Yaskawa INFORM job: X2_55A(90,180).JBI

/JOB
//NAME X2_55A(90,180)
//POS
///NPOS 356,356,356,16,0,0
///TOOL 0
///POSTYPE PULSE
///PULSE
C00000=3109,-122452,-100913,-73,83322,449
C00001=-57547,-44507,-45529,-37768,86502,54365
C00002=-65928,-27646,-34572,-36764,84429,51561
C00003=-68932,-27355,-32037,-36417,82009,51120
C00004=-70133,-27145,-30956,-36281,81048,50940
C00005=-71251,-29014,-32241,-36126,80438,50675
C00006=-70937,-28647,-32231,-36159,80720,50713
C00007=-70939,-28348,-30359,-36244,79905,50983
C00008=-70850,-28266,-30689,-36235,80141,50942
C00009=-71777,-26040,-29151,-36077,79912,50630
C00010=-70850,-28266,-30689,-36235,80141,50942
C00011=-69640,-28520,-31799,-36368,81104,51127
C00012=-66609,-28920,-34410,-36705,83528,51580
C00013=-67283,-40522,-42778,-21836,57084,56863
C00014=-69666,-37175,-37764,-20920,55189,56238
C00015=-70593,-35779,-35703,-20558,54438,55990
C00016=-70595,-35399,-33785,-20806,53513,56182
C00017=-71439,-34878,-33636,-20299,53466,55818
C00018=-72039,-34449,-33357,-19958,53365,55574
C00019=-70600,-35459,-34012,-20775,53614,56158
C00020=-69673,-36879,-36092,-21134,54366,56408
C00021=-67291,-40287,-41153,-22043,56263,57036
C00022=-54757,-64654,-56678,-26574,55995,60610
C00023=-66125,-22240,-12046,-37767,75415,54591
C00024=-69120,-21153,-8852,-37720,72980,54160
C00025=-70318,-20628,-7503,-37704,72009,53986
C00026=-71434,-22405,-8777,-37615,71420,53709
C00027=-71106,-21887,-8483,-37633,71631,53777
C00028=-71108,-21030,-6132,-37829,70825,54070
C00029=-70936,-21522,-6647,-37833,70951,54100
C00030=-71862,-19395,-5114,-37710,70668,53794
C00031=-70936,-21522,-6647,-37833,70951,54100
C00032=-66696,-23294,-11311,-37869,74371,54717
C00033=-67477,-36863,-27706,-23811,50186,58383
C00034=-69851,-33011,-22248,-22972,48242,57743
C00035=-70774,-31410,-19999,-22642,47467,57490
C00036=-70776,-30665,-17785,-22990,46560,57721
C00037=-70660,-30833,-18099,-23019,46692,57745
C00038=-72095,-29866,-17454,-22146,46391,57112
C00039=-70660,-30833,-18099,-23019,46692,57745
C00040=-67358,-36360,-25881,-24167,49428,58637
C00041=-57529,-55156,-37288,-27679,48780,61381
C00042=-66162,-22086,-11962,-37760,75421,54573
C00043=-69154,-20998,-8767,-37712,72987,54143
C00044=-70350,-20473,-7417,-37696,72017,53969
C00045=-71465,-22250,-8693,-37606,71429,53692
C00046=-74636,-20949,-11222,-31484,73172,51606
C00047=-71188,-20903,-6014,-37823,70785,54049
C00048=-71042,-21313,-6495,-37820,70916,54065
C00049=-71965,-19182,-4958,-37697,70633,53761
C00050=-71042,-21313,-6495,-37820,70916,54065
C00051=-66808,-23094,-11168,-37857,74333,54682
C00052=-67549,-36655,-27551,-23768,50176,58352
C00053=-69918,-32800,-22087,-22931,48232,57713
C00054=-70839,-31198,-19836,-22602,47457,57461
C00055=-70841,-30454,-17622,-22950,46550,57692
C00056=-70807,-30574,-17946,-22919,46687,57673
C00057=-72239,-29602,-17296,-22048,46388,57041
C00058=-70807,-30574,-17946,-22919,46687,57673
C00059=-67516,-36108,-25740,-24067,49421,58563
C00060=-58006,-54475,-36914,-27392,48730,61159
C00061=-66150,-22232,-11999,-37769,75384,54591
C00062=-69146,-21141,-8802,-37722,72949,54160
C00063=-70343,-20614,-7451,-37706,71978,53986
C00064=-71460,-22391,-8725,-37617,71389,53709
C00065=-76354,-9489,-5358,-27324,81880,47708
C00066=-80283,-13253,-8650,-21924,78677,47540
C00067=-72863,-23243,-10183,-35045,70283,54216
C00068=-72091,-18996,-4868,-37675,70611,53714
C00069=-71171,-21130,-6410,-37799,70893,54017
C00070=-66943,-22922,-11092,-37839,74307,54632
C00071=-67592,-36530,-27454,-23743,50168,58333
C00072=-69958,-32673,-21987,-22907,48224,57696
C00073=-70878,-31070,-19735,-22578,47450,57444
C00074=-70881,-30326,-17520,-22926,46541,57675
C00075=-70888,-30451,-17880,-22864,46685,57634
C00076=-72318,-29476,-17227,-21993,46388,57002
C00077=-70888,-30451,-17880,-22864,46685,57634
C00078=-67602,-35989,-25679,-24012,49417,58523
C00079=-55368,-59030,-40465,-28749,49477,62233
C00080=-66281,-21711,-11569,-37757,75329,54554
C00081=-69266,-20611,-8362,-37710,72898,54126
C00082=-75255,-19909,-10818,-29439,72911,51436
C00083=-75255,-19389,-9203,-29543,72275,51605
C00084=-75255,-19909,-10818,-29439,72911,51436
C00085=-76150,-21069,-11659,-29326,72528,51179
C00086=-75255,-19909,-10818,-29439,72911,51436
C00087=-75952,-17840,-9303,-29323,72782,51192
C00088=-76627,-15764,-7759,-29212,72649,50956
C00089=-75952,-17840,-9303,-29323,72782,51192
C00090=-67008,-22654,-10922,-37828,74305,54605
C00091=-67726,-36243,-27274,-23659,50164,58271
C00092=-70084,-32383,-21799,-22824,48221,57636
C00093=-71001,-30778,-19544,-22496,47446,57385
C00094=-71004,-30035,-17329,-22843,46537,57615
C00095=-71019,-30169,-17685,-22780,46672,57573
C00096=-72445,-29190,-17028,-21910,46377,56942
C00097=-71019,-30169,-17685,-22780,46672,57573
C00098=-67743,-35714,-25496,-23926,49403,58459
C00099=-55737,-58548,-40210,-28536,49431,62065
C00100=-62068,-51424,-36574,-22006,75894,31841
C00101=-60714,-28502,-21418,-45365,79926,-4626
C00102=-66771,-18477,-14837,-68384,79212,-42474
C00103=-69189,-16510,-10390,-68595,76911,-42051
C00104=-70947,-14387,-8158,-68595,75621,-42165
C00105=-70947,-13867,-6433,-68771,75311,-41816
C00106=-70947,-14164,-7409,-68671,75485,-42013
C00107=-71934,-13328,-6772,-68630,74836,-42164
C00108=-70947,-14164,-7409,-68671,75485,-42013
C00109=-66757,-18118,-13479,-68487,78967,-42191
C00110=-63228,-11986,-9955,-68477,81724,-42141
C00111=-63445,-12696,-10506,-68473,81568,-42159
C00112=-66764,-18741,-15037,-68386,79212,-42468
C00113=-69186,-16774,-10592,-68597,76909,-42046
C00114=-70875,-13966,-7307,-68664,75547,-42021
C00115=-70875,-13696,-6414,-68755,75387,-41841
C00116=-70875,-13966,-7307,-68664,75547,-42021
C00117=-71778,-13120,-6662,-68624,74954,-42161
C00118=-70875,-13966,-7307,-68664,75547,-42021
C00119=-66661,-18411,-13691,-68493,79023,-42169
C00120=-63445,-12696,-10506,-68473,81568,-42159
C00121=-63865,-13952,-11469,-68464,81265,-42192
C00122=-66537,-18783,-15074,-68396,79365,-42438
C00123=-68961,-16831,-10641,-68604,77060,-42016
C00124=-70699,-13899,-7235,-68671,75661,-41992
C00125=-70699,-13580,-6183,-68778,75474,-41781
C00126=-70699,-13899,-7235,-68671,75661,-41992
C00127=-71619,-12932,-6499,-68632,75061,-42136
C00128=-70699,-13899,-7235,-68671,75661,-41992
C00129=-66539,-18412,-13687,-68498,79104,-42151
C00130=-63865,-13952,-11469,-68464,81265,-42192
C00131=-63260,-13360,-10989,-68484,81675,-42115
C00132=-66441,-19168,-15326,-68406,79413,-42406
C00133=-68872,-17218,-10898,-68615,77104,-41986
C00134=-70768,-14438,-7612,-68680,75597,-41981
C00135=-70768,-14095,-6488,-68794,75397,-41755
C00136=-70768,-14438,-7612,-68680,75597,-41981
C00137=-71628,-14065,-7329,-68648,75028,-42105
C00138=-70768,-14438,-7612,-68680,75597,-41981
C00139=-66448,-18790,-13996,-68502,79163,-42137
C00140=-63260,-13360,-10989,-68484,81675,-42115
C00141=-61191,-13759,-10892,-73705,82833,-41510
C00142=-64290,-19711,-15321,-73681,80576,-41688
C00143=-66947,-17907,-11278,-73881,78250,-41270
C00144=-68815,-15776,-8601,-73968,76784,-41217
C00145=-68815,-15434,-7486,-74073,76629,-40986
C00146=-68815,-15776,-8601,-73968,76784,-41217
C00147=-69853,-15286,-8234,-73951,76069,-41336
C00148=-68815,-15776,-8601,-73968,76784,-41217
C00149=-64280,-19397,-14090,-73763,80400,-41421
C00150=-61191,-13759,-10892,-73705,82833,-41510
C00151=-66549,4585,8841,-68757,84788,-39990
C00152=-68719,6226,13286,-68971,82600,-39461
C00153=-70299,8854,16372,-69091,81328,-39429
C00154=-70565,4457,12550,-69090,81182,-39506
C00155=-70671,1948,10411,-69092,81122,-39532
C00156=-70937,-1261,7725,-69102,80944,-39568
C00157=-71174,-3897,5579,-69114,80771,-39582
C00158=-71415,-5667,4175,-69128,80592,-39593
C00159=-71589,-7772,2495,-69141,80458,-39594
C00160=-69844,-9224,758,-68895,80432,-50090
C00161=-67406,-9976,-2757,-68634,82758,-50534
C00162=-64294,-4174,1857,-68554,84904,-50183
C00163=-64639,7717,11547,-68707,86051,-39715
C00164=-66369,4107,8421,-68752,84915,-39972
C00165=-68544,5733,12848,-68963,82723,-39446
C00166=-70109,8786,16479,-69096,81419,-39361
C00167=-70297,4081,12289,-69084,81351,-39454
C00168=-70614,-406,8517,-69095,81102,-39512
C00169=-70890,-3195,6296,-69112,80891,-39521
C00170=-71255,-5626,4463,-69140,80599,-39517
C00171=-71566,-7424,3025,-69158,80374,-39541
C00172=-69656,-9705,371,-68890,80554,-50061
C00173=-67211,-10445,-3132,-68632,82884,-50504
C00174=-63438,-3299,2558,-68529,85486,-50077
C00175=-64904,8869,12572,-68717,85859,-39734
C00176=-66728,5060,9252,-68761,84665,-40010
C00177=-68892,6716,13713,-68979,82479,-39479
C00178=-70477,9030,16462,-69095,81221,-39469
C00179=-70621,5852,13649,-69089,81161,-39530
C00180=-70741,3427,11502,-69084,81107,-39575
C00181=-70957,-7,8601,-69089,80968,-39614
C00182=-71235,-3202,5925,-69097,80786,-39652
C00183=-71489,-5726,3878,-69109,80600,-39671
C00184=-71754,-7118,2931,-69135,80371,-39649
C00185=-70030,-8747,1134,-68898,80312,-50120
C00186=-67598,-9511,-2391,-68636,82634,-50565
C00187=-63663,-2057,3588,-68535,85336,-50109
C00188=-63900,9785,13379,-68685,86523,-39590
C00189=-66459,4347,8637,-68754,84850,-39980
C00190=-68632,5981,13072,-68967,82660,-39452
C00191=-70228,9427,16889,-69090,81369,-39412
C00192=-70256,7516,15203,-69086,81369,-39438
C00193=-70584,2390,10785,-69088,81181,-39517
C00194=-70847,-1463,7557,-69098,81005,-39554
C00195=-71203,-4827,4861,-69120,80739,-39570
C00196=-71527,-7834,2455,-69140,80496,-39585
C00197=-69750,-9463,570,-68893,80492,-50074
C00198=-67309,-10209,-2939,-68633,82820,-50518
C00199=-63863,-3734,2214,-68542,85196,-50129
C00200=-63361,11899,15268,-68667,86856,-39487
C00201=-66639,4823,9047,-68759,84726,-40000
C00202=-68806,6472,13500,-68975,82539,-39470
C00203=-70371,9492,16754,-69084,81316,-39482
C00204=-70406,7614,14987,-69071,81339,-39541
C00205=-70815,1914,10234,-69086,81061,-39593
C00206=-71160,-1949,7032,-69099,80826,-39630
C00207=-71480,-5381,4180,-69113,80607,-39668
C00208=-71698,-7658,2398,-69130,80431,-39664
C00209=-69937,-8985,946,-68896,80372,-50105
C00210=-67502,-9743,-2574,-68635,82696,-50550
C00211=-63039,-1186,4305,-68516,85757,-50029
C00212=-63804,-15836,-24938,-33383,81044,-33833
C00213=-63258,-44242,-52787,-23373,87348,-17537
C00214=-45457,-61378,-31703,-56361,46356,83670
C00215=-63650,-43074,-25993,-45661,44798,82564
C00216=-66314,-39383,-20678,-45469,42464,82291
C00217=-66918,-36654,-17674,-45533,41839,82291
C00218=-66822,-35437,-16825,-45503,41961,82277
C00219=-66732,-35006,-16524,-45511,42032,82290
C00220=-64645,-31599,-14317,-48183,45887,84406
C00221=-64296,-29134,-12669,-48119,46248,84396
C00222=-63820,-26748,-11175,-48100,46707,84404
C00223=-63109,-29591,-14333,-48037,47414,84404
C00224=-60528,-32714,-19448,-47978,49839,84498
C00225=-67866,-18058,-8941,-23337,65103,48953
C00226=-70222,-15115,-3728,-23038,62877,48478
C00227=-71019,-12738,-845,-22932,62145,48310
C00228=-72616,-17245,-4255,-21172,60226,46085
C00229=-73616,-20397,-6483,-20913,59741,45771
C00230=-73982,-21396,-7198,-20816,59580,45652
C00231=-72782,-13420,-2650,-23032,68738,42765
C00232=-71424,-14381,-4450,-23190,69684,43097
C00233=-69030,-17053,-9428,-23386,71918,43563
C00234=-69362,-15034,-7208,-34893,81212,68979
C00235=-71754,-15466,-4606,-34965,78725,68783
C00236=-72600,-16194,-3925,-35016,77725,68752
C00237=-74033,-12291,-1030,-34922,77318,68288
C00238=-74317,-11546,-458,-34905,77227,68199
C00239=-74455,-14836,-1302,-37403,72119,67993
C00240=-73330,-15101,-2651,-37376,73163,68109
C00241=-70777,-15355,-5703,-37313,75672,68325
C00242=-64737,-39088,-25802,-40098,74682,69478
C00243=-53091,-60542,-45293,-47415,47642,80398
C00244=-63422,-47376,-37973,-42415,48686,80430
C00245=-66097,-44034,-33002,-41935,46389,80068
C00246=-66682,-41433,-30082,-41934,45762,80055
C00247=-66426,-39531,-28938,-41893,46090,80031
C00248=-66144,-37902,-27886,-41909,46370,80051
C00249=-65467,-34288,-25654,-41944,47058,80086
C00250=-62899,-33876,-26604,-44822,51283,82174
C00251=-60308,-36583,-31327,-45053,53688,82354
C00252=-67726,-23407,-36448,-21685,78297,46429
C00253=-70089,-21663,-32282,-21173,76131,45959
C00254=-70847,-19835,-29787,-21017,75382,45815
C00255=-72612,-24426,-33008,-19186,73418,43731
C00256=-73313,-26973,-34814,-18991,73073,43530
C00257=-73750,-28127,-35541,-18872,72835,43409
C00258=-72685,-19752,-30962,-21756,81921,40284
C00259=-71295,-20339,-32550,-22004,82916,40605
C00260=-68894,-21809,-36497,-22419,85109,41062
C00261=-69210,-19992,-31537,-34666,91587,65802
C00262=-71606,-21576,-29855,-34416,89087,65610
C00263=-72545,-22706,-29436,-34329,88011,65563
C00264=-73736,-19082,-26828,-34209,87746,65164
C00265=-73876,-19138,-26700,-34340,87246,65092
C00266=-74191,-22242,-27567,-35926,82262,64646
C00267=-73185,-21848,-28433,-36023,83286,64728
C00268=-70628,-21004,-30580,-36304,85789,64959
C00269=-63500,-41614,-43915,-39144,82937,66913
C00270=-51083,-55789,-28797,-53955,43738,77608
C00271=-63909,-42641,-25730,-45502,44710,82450
C00272=-66558,-38941,-20402,-45309,42381,82178
C00273=-67126,-36171,-17521,-45309,41847,82142
C00274=-67034,-35116,-16750,-45307,41938,82145
C00275=-66872,-34228,-16138,-45314,42077,82163
C00276=-64623,-29682,-13170,-47994,46090,84285
C00277=-64367,-28039,-12066,-47957,46341,84285
C00278=-64141,-26180,-10783,-47945,46572,84281
C00279=-63346,-29164,-14043,-47920,47316,84312
C00280=-60776,-32299,-19172,-47861,49737,84405
C00281=-68069,-17598,-8601,-23280,65070,48879
C00282=-70417,-14643,-3372,-22982,62844,48406
C00283=-71449,-10477,1221,-22838,61926,48182
C00284=-73498,-15799,-2776,-20937,59845,45801
C00285=-74336,-18361,-4626,-20710,59468,45532
C00286=-74806,-19783,-5679,-20581,59274,45375
C00287=-73116,-10825,-379,-22979,68584,42666
C00288=-71613,-13902,-4086,-23153,69651,43031
C00289=-69228,-16586,-9079,-23349,71885,43493
C00290=-69547,-14561,-6882,-34883,81172,68916
C00291=-71934,-14986,-4277,-34953,78688,68720
C00292=-72986,-13222,-1607,-34989,77647,68617
C00293=-73715,-11547,-247,-34949,77364,68403
C00294=-74925,-8670,2089,-35073,76570,68005
C00295=-74789,-12370,664,-37364,72021,67879
C00296=-73505,-14616,-2317,-37354,73122,68047
C00297=-70959,-14879,-5376,-37292,75628,68262
C00298=-65183,-36967,-21616,-40314,73326,69808
C00299=-53228,-53274,-27436,-52865,42800,79914
C00300=-63520,-43290,-26124,-45740,44843,82622
C00301=-66190,-39604,-20816,-45549,42506,82348
C00302=-66900,-36698,-17594,-45598,41796,82332
C00303=-66609,-35418,-16854,-45581,42087,82339
C00304=-66490,-34479,-16216,-45562,42214,82337
C00305=-64381,-30847,-13853,-48196,46099,84439
C00306=-64009,-28704,-12465,-48169,46466,84442
C00307=-63758,-26820,-11226,-48128,46737,84427
C00308=-62989,-29805,-14477,-48096,47463,84450
C00309=-60403,-32922,-19585,-48036,49890,84545
C00310=-67763,-18288,-9111,-23365,65119,48991
C00311=-70125,-15350,-3906,-23066,62893,48514
C00312=-70717,-13403,-1445,-23008,62257,48410
C00313=-72577,-17861,-4625,-21199,60154,46117
C00314=-73271,-20124,-6266,-21016,59837,45895
C00315=-73854,-21888,-7506,-20866,59553,45712
C00316=-72474,-13787,-2972,-23087,68832,42865
C00317=-71329,-14621,-4631,-23208,69700,43131
C00318=-68930,-17287,-9602,-23404,71934,43598
C00319=-69254,-15266,-7415,-34896,81263,69008
C00320=-71649,-15705,-4819,-34968,78775,68810
C00321=-72477,-16320,-4101,-35016,77809,68777
C00322=-73799,-12901,-1530,-34934,77409,68356
C00323=-74042,-12557,-1142,-35120,76926,68260
C00324=-74352,-14974,-1438,-37409,72173,68017
C00325=-73226,-15345,-2868,-37384,73214,68135
C00326=-70671,-15592,-5914,-37320,75725,68353
C00327=-62836,-37760,-18291,-40933,72527,71194
C00328=-50354,-56570,-29213,-54300,44067,82652
C00329=-63780,-42857,-25862,-45581,44754,82507
C00330=-66436,-39162,-20540,-45388,42422,82235
C00331=-67179,-36421,-17487,-45403,41711,82196
C00332=-66965,-35184,-16697,-45393,41923,82201
C00333=-64496,-29723,-13207,-48023,46159,84319
C00334=-64008,-26353,-10886,-48014,46622,84337
C00335=-63228,-29377,-14188,-47979,47365,84358
C00336=-60652,-32506,-19310,-47920,49788,84451
C00337=-67968,-17828,-8771,-23308,65086,48916
C00338=-70320,-14879,-3550,-23010,62860,48442
C00339=-71178,-12230,-319,-22903,62044,48268
C00340=-72994,-16926,-3771,-21083,60004,45976
C00341=-73940,-20147,-6136,-20831,59579,45672
C00342=-74304,-21288,-6996,-20731,59435,45550
C00343=-72900,-12965,-2204,-23017,68666,42732
C00344=-71519,-14141,-4268,-23172,69668,43064
C00345=-69129,-16819,-9253,-23368,71902,43528
C00346=-69450,-14796,-7060,-34888,81202,68946
C00347=-71839,-15226,-4457,-34958,78717,68750
C00348=-72721,-15820,-3696,-35004,77716,68705
C00349=-73957,-12367,-1093,-34926,77347,68309
C00350=-74315,-11825,-532,-35105,76814,68183
C00351=-74587,-14424,-1021,-37384,72093,67943
C00352=-73412,-14859,-2501,-37364,73153,68076
C00353=-70864,-15116,-5555,-37302,75660,68292
C00354=-61264,-35992,-20137,-38019,78448,71435
C00355=3322,-122452,-100913,-73,83322,449
BC00000=198923,666220,911653
BC00001=345030,666220,1075175
BC00002=345030,666220,1075175
BC00003=345030,666220,1075175
BC00004=345030,666220,1075175
BC00005=345030,666220,1075175
BC00006=345030,666220,1075175
BC00007=345030,666220,1075175
BC00008=345030,666220,1075175
BC00009=345030,666220,1075175
BC00010=345030,666220,1075175
BC00011=345030,666220,1075175
BC00012=345030,666220,1075175
BC00013=320007,666220,1075175
BC00014=320007,666220,1075175
BC00015=320007,666220,1075175
BC00016=320007,666220,1075175
BC00017=320007,666220,1075175
BC00018=320007,666220,1075175
BC00019=320007,666220,1075175
BC00020=320007,666220,1075175
BC00021=320007,666220,1075175
BC00022=314803,666681,1075175
BC00023=345023,666220,1034707
BC00024=345023,666220,1034707
BC00025=345023,666220,1034707
BC00026=345023,666220,1034707
BC00027=345023,666220,1034707
BC00028=345023,666220,1034707
BC00029=345023,666220,1034707
BC00030=345023,666220,1034707
BC00031=345023,666220,1034707
BC00032=345023,666220,1034707
BC00033=320036,666220,995579
BC00034=320036,666220,995579
BC00035=320036,666220,995579
BC00036=320036,666220,995579
BC00037=320036,666220,995579
BC00038=320036,666220,995579
BC00039=320036,666220,995579
BC00040=320036,666220,995579
BC00041=314838,666681,1004817
BC00042=344960,666220,872758
BC00043=344960,666220,872758
BC00044=344960,666220,872758
BC00045=344960,666220,872758
BC00046=344960,666220,872758
BC00047=344960,666220,872758
BC00048=344960,666220,872758
BC00049=344960,666220,872758
BC00050=344960,666220,872758
BC00051=344960,666220,872758
BC00052=320210,666220,833606
BC00053=320210,666220,833606
BC00054=320210,666220,833606
BC00055=320210,666220,833606
BC00056=320210,666220,833606
BC00057=320210,666220,833606
BC00058=320210,666220,833606
BC00059=320210,666220,833606
BC00060=314872,666681,843515
BC00061=345087,666220,710509
BC00062=345087,666220,710509
BC00063=345087,666220,710509
BC00064=345087,666220,710509
BC00065=345087,666220,710509
BC00066=345087,666220,710509
BC00067=345087,666220,710509
BC00068=345087,666220,710509
BC00069=345087,666220,710509
BC00070=345087,666220,710509
BC00071=320046,666220,671597
BC00072=320046,666220,671597
BC00073=320046,666220,671597
BC00074=320046,666220,671597
BC00075=320046,666220,671597
BC00076=320046,666220,671597
BC00077=320046,666220,671597
BC00078=320046,666220,671597
BC00079=314907,666681,682214
BC00080=344913,666220,548992
BC00081=344913,666220,548992
BC00082=344913,666220,548992
BC00083=344913,666220,548992
BC00084=344913,666220,548992
BC00085=344913,666220,548992
BC00086=344913,666220,548992
BC00087=344913,666220,548992
BC00088=344913,666220,548992
BC00089=344913,666220,548992
BC00090=344913,666220,548992
BC00091=320171,666220,510267
BC00092=320171,666220,510267
BC00093=320171,666220,510267
BC00094=320171,666220,510267
BC00095=320171,666220,510267
BC00096=320171,666220,510267
BC00097=320171,666220,510267
BC00098=320171,666220,510267
BC00099=314942,666681,520912
BC00100=378648,679076,578921
BC00101=388411,672648,490370
BC00102=398174,666220,401819
BC00103=398174,666220,401819
BC00104=398174,666220,401819
BC00105=398174,666220,401819
BC00106=398174,666220,401819
BC00107=398174,666220,401819
BC00108=398174,666220,401819
BC00109=398174,666220,401819
BC00110=398174,666220,401819
BC00111=398174,666220,563089
BC00112=398174,666220,563089
BC00113=398174,666220,563089
BC00114=398174,666220,563089
BC00115=398174,666220,563089
BC00116=398174,666220,563089
BC00117=398174,666220,563089
BC00118=398174,666220,563089
BC00119=398174,666220,563089
BC00120=398174,666220,563089
BC00121=398174,666220,725161
BC00122=398174,666220,725161
BC00123=398174,666220,725161
BC00124=398174,666220,725161
BC00125=398174,666220,725161
BC00126=398174,666220,725161
BC00127=398174,666220,725161
BC00128=398174,666220,725161
BC00129=398174,666220,725161
BC00130=398174,666220,725161
BC00131=398174,666220,887461
BC00132=398174,666220,887461
BC00133=398174,666220,887461
BC00134=398174,666220,887461
BC00135=398174,666220,887461
BC00136=398174,666220,887461
BC00137=398174,666220,887461
BC00138=398174,666220,887461
BC00139=398174,666220,887461
BC00140=398174,666220,887461
BC00141=398174,666220,1018524
BC00142=398174,666220,1018524
BC00143=398174,666220,1018524
BC00144=398174,666220,1018524
BC00145=398174,666220,1018524
BC00146=398174,666220,1018524
BC00147=398174,666220,1018524
BC00148=398174,666220,1018524
BC00149=398174,666220,1018524
BC00150=398174,666220,1018524
BC00151=398174,666220,750812
BC00152=398174,666220,750812
BC00153=398174,666220,750812
BC00154=398174,666220,750812
BC00155=398174,666220,750812
BC00156=398174,666220,750812
BC00157=398174,666220,750812
BC00158=398174,666220,750812
BC00159=398174,666220,750812
BC00160=398174,666220,750812
BC00161=398174,666220,750812
BC00162=398174,666220,750812
BC00163=398174,666220,1074971
BC00164=398174,666220,1074971
BC00165=398174,666220,1074971
BC00166=398174,666220,1074971
BC00167=398174,666220,1074971
BC00168=398174,666220,1074971
BC00169=398174,666220,1074971
BC00170=398174,666220,1074971
BC00171=398174,666220,1074971
BC00172=398174,666220,1074971
BC00173=398174,666220,1074971
BC00174=398174,666220,1074971
BC00175=398174,666220,427406
BC00176=398174,666220,427406
BC00177=398174,666220,427406
BC00178=398174,666220,427406
BC00179=398174,666220,427406
BC00180=398174,666220,427406
BC00181=398174,666220,427406
BC00182=398174,666220,427406
BC00183=398174,666220,427406
BC00184=398174,666220,427406
BC00185=398174,666220,427406
BC00186=398174,666220,427406
BC00187=398174,666220,427406
BC00188=398174,666220,912918
BC00189=398174,666220,912918
BC00190=398174,666220,912918
BC00191=398174,666220,912918
BC00192=398174,666220,912918
BC00193=398174,666220,912918
BC00194=398174,666220,912918
BC00195=398174,666220,912918
BC00196=398174,666220,912918
BC00197=398174,666220,912918
BC00198=398174,666220,912918
BC00199=398174,666220,912918
BC00200=398174,666220,588706
BC00201=398174,666220,588706
BC00202=398174,666220,588706
BC00203=398174,666220,588706
BC00204=398174,666220,588706
BC00205=398174,666220,588706
BC00206=398174,666220,588706
BC00207=398174,666220,588706
BC00208=398174,666220,588706
BC00209=398174,666220,588706
BC00210=398174,666220,588706
BC00211=398174,666220,588706
BC00212=398174,666681,626567
BC00213=360198,666681,720930
BC00214=313360,666681,837312
BC00215=325296,666220,810137
BC00216=325296,666220,810137
BC00217=325296,666220,810137
BC00218=325296,666220,810137
BC00219=325296,666220,810137
BC00220=325296,666220,810137
BC00221=325296,666220,810137
BC00222=325296,666220,810137
BC00223=325296,666220,810137
BC00224=325296,666220,810137
BC00225=319313,666220,902547
BC00226=319313,666220,902547
BC00227=319313,666220,902547
BC00228=319313,666220,902547
BC00229=319313,666220,902547
BC00230=319313,666220,902547
BC00231=319313,666220,902547
BC00232=319313,666220,902547
BC00233=319313,666220,902547
BC00234=349969,666220,883404
BC00235=349969,666220,883404
BC00236=349969,666220,883404
BC00237=349969,666220,883404
BC00238=349969,666220,883404
BC00239=349969,666220,883404
BC00240=349969,666220,883404
BC00241=349969,666220,883404
BC00242=354755,666681,897949
BC00243=313290,666681,1075175
BC00244=325290,666220,1075175
BC00245=325290,666220,1075175
BC00246=325290,666220,1075175
BC00247=325290,666220,1075175
BC00248=325290,666220,1075175
BC00249=325290,666220,1075175
BC00250=325290,666220,1075175
BC00251=325290,666220,1075175
BC00252=319307,666220,1075175
BC00253=319307,666220,1075175
BC00254=319307,666220,1075175
BC00255=319307,666220,1075175
BC00256=319307,666220,1075175
BC00257=319307,666220,1075175
BC00258=319307,666220,1075175
BC00259=319307,666220,1075175
BC00260=319307,666220,1075175
BC00261=349934,666220,1075175
BC00262=349934,666220,1075175
BC00263=349934,666220,1075175
BC00264=349934,666220,1075175
BC00265=349934,666220,1075175
BC00266=349934,666220,1075175
BC00267=349934,666220,1075175
BC00268=349934,666220,1075175
BC00269=354685,666681,1075175
BC00270=313430,666681,513902
BC00271=325303,666220,486731
BC00272=325303,666220,486731
BC00273=325303,666220,486731
BC00274=325303,666220,486731
BC00275=325303,666220,486731
BC00276=325303,666220,486731
BC00277=325303,666220,486731
BC00278=325303,666220,486731
BC00279=325303,666220,486731
BC00280=325303,666220,486731
BC00281=319320,666220,579141
BC00282=319320,666220,579141
BC00283=319320,666220,579141
BC00284=319320,666220,579141
BC00285=319320,666220,579141
BC00286=319320,666220,579141
BC00287=319320,666220,579141
BC00288=319320,666220,579141
BC00289=319320,666220,579141
BC00290=349947,666220,559795
BC00291=349947,666220,559795
BC00292=349947,666220,559795
BC00293=349947,666220,559795
BC00294=349947,666220,559795
BC00295=349947,666220,559795
BC00296=349947,666220,559795
BC00297=349947,666220,559795
BC00298=354825,666681,574539
BC00299=313325,666681,999420
BC00300=325293,666220,972243
BC00301=325293,666220,972243
BC00302=325293,666220,972243
BC00303=325293,666220,972243
BC00304=325293,666220,972243
BC00305=325293,666220,972243
BC00306=325293,666220,972243
BC00307=325293,666220,972243
BC00308=325293,666220,972243
BC00309=325293,666220,972243
BC00310=319310,666220,1064653
BC00311=319310,666220,1064653
BC00312=319310,666220,1064653
BC00313=319310,666220,1064653
BC00314=319310,666220,1064653
BC00315=319310,666220,1064653
BC00316=319310,666220,1064653
BC00317=319310,666220,1064653
BC00318=319310,666220,1064653
BC00319=349937,666220,1045308
BC00320=349937,666220,1045308
BC00321=349937,666220,1045308
BC00322=349937,666220,1045308
BC00323=349937,666220,1045308
BC00324=349937,666220,1045308
BC00325=349937,666220,1045308
BC00326=349937,666220,1045308
BC00327=354720,666681,1060057
BC00328=313395,666681,675204
BC00329=325299,666220,648031
BC00330=325299,666220,648031
BC00331=325299,666220,648031
BC00332=325299,666220,648031
BC00333=325299,666220,648031
BC00334=325299,666220,648031
BC00335=325299,666220,648031
BC00336=325299,666220,648031
BC00337=319316,666220,740441
BC00338=319316,666220,740441
BC00339=319316,666220,740441
BC00340=319316,666220,740441
BC00341=319316,666220,740441
BC00342=319316,666220,740441
BC00343=319316,666220,740441
BC00344=319316,666220,740441
BC00345=319316,666220,740441
BC00346=349944,666220,721095
BC00347=349944,666220,721095
BC00348=349944,666220,721095
BC00349=349944,666220,721095
BC00350=349944,666220,721095
BC00351=349944,666220,721095
BC00352=349944,666220,721095
BC00353=349944,666220,721095
BC00354=349944,666220,721095
BC00355=87761,666220,1075229
EC00000=798156,1112951
EC00001=798156,1112951
EC00002=798156,1112951
EC00003=798156,1112951
EC00004=798156,1112951
EC00005=798156,1112951
EC00006=798156,1112951
EC00007=798156,1112951
EC00008=798156,1112951
EC00009=798156,1112951
EC00010=798156,1112951
EC00011=798156,1112951
EC00012=798156,1112951
EC00013=798156,1112951
EC00014=798156,1112951
EC00015=798156,1112951
EC00016=798156,1112951
EC00017=798156,1112951
EC00018=798156,1112951
EC00019=798156,1112951
EC00020=798156,1112951
EC00021=798156,1112951
EC00022=798156,1112951
EC00023=798156,1112951
EC00024=798156,1112951
EC00025=798156,1112951
EC00026=798156,1112951
EC00027=798156,1112951
EC00028=798156,1112951
EC00029=798156,1112951
EC00030=798156,1112951
EC00031=798156,1112951
EC00032=798156,1112951
EC00033=798156,1112951
EC00034=798156,1112951
EC00035=798156,1112951
EC00036=798156,1112951
EC00037=798156,1112951
EC00038=798156,1112951
EC00039=798156,1112951
EC00040=798156,1112951
EC00041=798156,1112951
EC00042=798156,1112951
EC00043=798156,1112951
EC00044=798156,1112951
EC00045=798156,1112951
EC00046=798156,1112951
EC00047=798156,1112951
EC00048=798156,1112951
EC00049=798156,1112951
EC00050=798156,1112951
EC00051=798156,1112951
EC00052=798156,1112951
EC00053=798156,1112951
EC00054=798156,1112951
EC00055=798156,1112951
EC00056=798156,1112951
EC00057=798156,1112951
EC00058=798156,1112951
EC00059=798156,1112951
EC00060=798156,1112951
EC00061=798156,1112951
EC00062=798156,1112951
EC00063=798156,1112951
EC00064=798156,1112951
EC00065=798156,1112951
EC00066=798156,1112951
EC00067=798156,1112951
EC00068=798156,1112951
EC00069=798156,1112951
EC00070=798156,1112951
EC00071=798156,1112951
EC00072=798156,1112951
EC00073=798156,1112951
EC00074=798156,1112951
EC00075=798156,1112951
EC00076=798156,1112951
EC00077=798156,1112951
EC00078=798156,1112951
EC00079=798156,1112951
EC00080=798156,1112951
EC00081=798156,1112951
EC00082=798156,1112951
EC00083=798156,1112951
EC00084=798156,1112951
EC00085=798156,1112951
EC00086=798156,1112951
EC00087=798156,1112951
EC00088=798156,1112951
EC00089=798156,1112951
EC00090=798156,1112951
EC00091=798156,1112951
EC00092=798156,1112951
EC00093=798156,1112951
EC00094=798156,1112951
EC00095=798156,1112951
EC00096=798156,1112951
EC00097=798156,1112951
EC00098=798156,1112951
EC00099=798156,1112951
EC00100=798156,1112951
EC00101=798156,1112951
EC00102=798156,1112951
EC00103=798156,1112951
EC00104=798156,1112951
EC00105=798156,1112951
EC00106=798156,1112951
EC00107=798156,1112951
EC00108=798156,1112951
EC00109=798156,1112951
EC00110=798156,1112951
EC00111=798156,1112951
EC00112=798156,1112951
EC00113=798156,1112951
EC00114=798156,1112951
EC00115=798156,1112951
EC00116=798156,1112951
EC00117=798156,1112951
EC00118=798156,1112951
EC00119=798156,1112951
EC00120=798156,1112951
EC00121=798156,1112951
EC00122=798156,1112951
EC00123=798156,1112951
EC00124=798156,1112951
EC00125=798156,1112951
EC00126=798156,1112951
EC00127=798156,1112951
EC00128=798156,1112951
EC00129=798156,1112951
EC00130=798156,1112951
EC00131=798156,1112951
EC00132=798156,1112951
EC00133=798156,1112951
EC00134=798156,1112951
EC00135=798156,1112951
EC00136=798156,1112951
EC00137=798156,1112951
EC00138=798156,1112951
EC00139=798156,1112951
EC00140=798156,1112951
EC00141=798156,1112951
EC00142=798156,1112951
EC00143=798156,1112951
EC00144=798156,1112951
EC00145=798156,1112951
EC00146=798156,1112951
EC00147=798156,1112951
EC00148=798156,1112951
EC00149=798156,1112951
EC00150=798156,1112951
EC00151=798156,1112951
EC00152=798156,1112951
EC00153=798156,1112951
EC00154=798156,1112951
EC00155=798156,1112951
EC00156=798156,1112951
EC00157=798156,1112951
EC00158=798156,1112951
EC00159=798156,1112951
EC00160=798156,1112951
EC00161=798156,1112951
EC00162=798156,1112951
EC00163=798156,1112951
EC00164=798156,1112951
EC00165=798156,1112951
EC00166=798156,1112951
EC00167=798156,1112951
EC00168=798156,1112951
EC00169=798156,1112951
EC00170=798156,1112951
EC00171=798156,1112951
EC00172=798156,1112951
EC00173=798156,1112951
EC00174=798156,1112951
EC00175=798156,1112951
EC00176=798156,1112951
EC00177=798156,1112951
EC00178=798156,1112951
EC00179=798156,1112951
EC00180=798156,1112951
EC00181=798156,1112951
EC00182=798156,1112951
EC00183=798156,1112951
EC00184=798156,1112951
EC00185=798156,1112951
EC00186=798156,1112951
EC00187=798156,1112951
EC00188=798156,1112951
EC00189=798156,1112951
EC00190=798156,1112951
EC00191=798156,1112951
EC00192=798156,1112951
EC00193=798156,1112951
EC00194=798156,1112951
EC00195=798156,1112951
EC00196=798156,1112951
EC00197=798156,1112951
EC00198=798156,1112951
EC00199=798156,1112951
EC00200=798156,1112951
EC00201=798156,1112951
EC00202=798156,1112951
EC00203=798156,1112951
EC00204=798156,1112951
EC00205=798156,1112951
EC00206=798156,1112951
EC00207=798156,1112951
EC00208=798156,1112951
EC00209=798156,1112951
EC00210=798156,1112951
EC00211=798156,1112951
EC00212=798156,1112951
EC00213=798156,1112951
EC00214=798156,1112951
EC00215=798156,1112951
EC00216=798156,1112951
EC00217=798156,1112951
EC00218=798156,1112951
EC00219=798156,1112951
EC00220=798156,1112951
EC00221=798156,1112951
EC00222=798156,1112951
EC00223=798156,1112951
EC00224=798156,1112951
EC00225=798156,1112951
EC00226=798156,1112951
EC00227=798156,1112951
EC00228=798156,1112951
EC00229=798156,1112951
EC00230=798156,1112951
EC00231=798156,1112951
EC00232=798156,1112951
EC00233=798156,1112951
EC00234=798156,1112951
EC00235=798156,1112951
EC00236=798156,1112951
EC00237=798156,1112951
EC00238=798156,1112951
EC00239=798156,1112951
EC00240=798156,1112951
EC00241=798156,1112951
EC00242=798156,1112951
EC00243=798156,1112951
EC00244=798156,1112951
EC00245=798156,1112951
EC00246=798156,1112951
EC00247=798156,1112951
EC00248=798156,1112951
EC00249=798156,1112951
EC00250=798156,1112951
EC00251=798156,1112951
EC00252=798156,1112951
EC00253=798156,1112951
EC00254=798156,1112951
EC00255=798156,1112951
EC00256=798156,1112951
EC00257=798156,1112951
EC00258=798156,1112951
EC00259=798156,1112951
EC00260=798156,1112951
EC00261=798156,1112951
EC00262=798156,1112951
EC00263=798156,1112951
EC00264=798156,1112951
EC00265=798156,1112951
EC00266=798156,1112951
EC00267=798156,1112951
EC00268=798156,1112951
EC00269=798156,1112951
EC00270=798156,1112951
EC00271=798156,1112951
EC00272=798156,1112951
EC00273=798156,1112951
EC00274=798156,1112951
EC00275=798156,1112951
EC00276=798156,1112951
EC00277=798156,1112951
EC00278=798156,1112951
EC00279=798156,1112951
EC00280=798156,1112951
EC00281=798156,1112951
EC00282=798156,1112951
EC00283=798156,1112951
EC00284=798156,1112951
EC00285=798156,1112951
EC00286=798156,1112951
EC00287=798156,1112951
EC00288=798156,1112951
EC00289=798156,1112951
EC00290=798156,1112951
EC00291=798156,1112951
EC00292=798156,1112951
EC00293=798156,1112951
EC00294=798156,1112951
EC00295=798156,1112951
EC00296=798156,1112951
EC00297=798156,1112951
EC00298=798156,1112951
EC00299=798156,1112951
EC00300=798156,1112951
EC00301=798156,1112951
EC00302=798156,1112951
EC00303=798156,1112951
EC00304=798156,1112951
EC00305=798156,1112951
EC00306=798156,1112951
EC00307=798156,1112951
EC00308=798156,1112951
EC00309=798156,1112951
EC00310=798156,1112951
EC00311=798156,1112951
EC00312=798156,1112951
EC00313=798156,1112951
EC00314=798156,1112951
EC00315=798156,1112951
EC00316=798156,1112951
EC00317=798156,1112951
EC00318=798156,1112951
EC00319=798156,1112951
EC00320=798156,1112951
EC00321=798156,1112951
EC00322=798156,1112951
EC00323=798156,1112951
EC00324=798156,1112951
EC00325=798156,1112951
EC00326=798156,1112951
EC00327=798156,1112951
EC00328=798156,1112951
EC00329=798156,1112951
EC00330=798156,1112951
EC00331=798156,1112951
EC00332=798156,1112951
EC00333=798156,1112951
EC00334=798156,1112951
EC00335=798156,1112951
EC00336=798156,1112951
EC00337=798156,1112951
EC00338=798156,1112951
EC00339=798156,1112951
EC00340=798156,1112951
EC00341=798156,1112951
EC00342=798156,1112951
EC00343=798156,1112951
EC00344=798156,1112951
EC00345=798156,1112951
EC00346=798156,1112951
EC00347=798156,1112951
EC00348=798156,1112951
EC00349=798156,1112951
EC00350=798156,1112951
EC00351=798156,1112951
EC00352=798156,1112951
EC00353=798156,1112951
EC00354=798156,1112951
EC00355=798156,1112951
///POSTYPE BASE
///RECTAN
///RCONF 0,0,0,0,0,0,0,0,0,0,0,0,0,0,0,0,0,0,0,0,0,0,0,0
P00006=0.222,-3.123,-1.508,0.0000,0.0000,0.0000
P00021=-0.225,-6.128,-0.405,0.0000,0.0000,0.0000
P00022=0.222,-3.123,-1.508,0.0000,0.0000,0.0000
P00023=0.143,-0.036,0.682,0.0000,0.0000,0.0000
P00031=1.853,-0.001,-1.549,0.0000,0.0000,0.0000
P00032=1.957,0.503,-7.217,0.0000,0.0000,0.0000
///RCONF 0,0,0,0,1,0,0,0,0,0,0,0,0,0,0,0,0,0,0,0,0,0,0,0
P00033=-0.123,0.612,-5.012,0.0000,0.0000,0.0000
///RCONF 0,0,0,0,0,0,0,0,0,0,0,0,0,0,0,0,0,0,0,0,0,0,0,0
P00041=0.192,3.924,0.305,0.0000,0.0000,0.0000
P00042=-0.217,1.941,0.413,0.0000,0.0000,0.0000
P00043=-0.044,-1.937,1.197,0.0000,0.0000,0.0000
P00051=0.367,3.892,0.009,0.0000,0.0000,0.0000
P00052=0.088,2.832,-0.342,0.0000,0.0000,0.0000
P00053=0.134,6.594,0.107,0.0000,0.0000,0.0000
P00061=1.575,-3.405,-0.752,0.0000,0.0000,0.0000
P00062=-0.135,-0.848,-1.706,0.0000,0.0000,0.0000
P00063=0.036,-0.654,-3.005,0.0000,0.0000,0.0000
//INST
///DATE 2025/02/19 15:11
///ATTR SC,RW
///GROUP1 RB1,BS1
///GROUP2 ST1
NOP
'X2_55a(90,180)
MOVJ C00000 BC00000 VJ=100.00  +MOVJ EC00000 VJ=100.00
MOVJ C00001 BC00001 VJ=100.00  +MOVJ EC00001 VJ=100.00
'Path S3757
SFTOF3D
MOVJ C00002 BC00002 VJ=100.00  +MOVJ EC00002 VJ=100.00
MOVL C00003 BC00003 V=800.0  +MOVJ EC00003 VJ=100.00
SMOVL C00004 BC00004 V=166.7  +MOVJ EC00004
SREFP 3 C00005 BC00005  +REFP EC00005
CALL JOB:SEARCH-R1-S13D
SET P021 P006
SFTON3D P021
SMOVL C00006 BC00006 V=166.7  +MOVJ EC00006
SREFP 3 C00007 BC00007  +REFP EC00007
CALL JOB:SEARCH-R1-S13D
SET P021 P006
SFTON3D P021
SMOVL C00008 BC00008 V=166.7  +MOVJ EC00008
SREFP 3 C00009 BC00009  +REFP EC00009
CALL JOB:SEARCH-R1-S13D
SET P021 P006
SFTON3D P021
SMOVL C00010 BC00010 V=166.7  +MOVJ EC00010
MOVL C00011 BC00011 V=800.0  +MOVJ EC00011 VJ=100.00
MOVL C00012 BC00012 V=1000.0  +MOVJ EC00012 VJ=100.00
'EndPath S3757
'Path S3758
SFTOF3D
MOVJ C00013 BC00013 VJ=100.00  +MOVJ EC00013 VJ=100.00
MOVL C00014 BC00014 V=800.0  +MOVJ EC00014 VJ=100.00
SMOVL C00015 BC00015 V=166.7  +MOVJ EC00015
SREFP 3 C00016 BC00016  +REFP EC00016
CALL JOB:SEARCH-R1-S13D
SET P022 P006
SFTON3D P022
SMOVL C00017 BC00017 V=166.7  +MOVJ EC00017
SREFP 3 C00018 BC00018  +REFP EC00018
CALL JOB:SEARCH-R1-S13D
SET P022 P006
SFTON3D P022
SMOVL C00019 BC00019 V=166.7  +MOVJ EC00019
MOVL C00020 BC00020 V=800.0  +MOVJ EC00020 VJ=100.00
MOVL C00021 BC00021 V=1000.0  +MOVJ EC00021 VJ=100.00
'EndPath S3758
MOVJ C00022 BC00022 VJ=100.00  +MOVJ EC00022 VJ=100.00
'
'Path S3759
SFTOF3D
MOVJ C00023 BC00023 VJ=100.00  +MOVJ EC00023 VJ=100.00
MOVL C00024 BC00024 V=800.0  +MOVJ EC00024 VJ=100.00
SMOVL C00025 BC00025 V=166.7  +MOVJ EC00025
SREFP 3 C00026 BC00026  +REFP EC00026
CALL JOB:SEARCH-R1-S13D
SET P031 P006
SFTON3D P031
SMOVL C00027 BC00027 V=166.7  +MOVJ EC00027
SREFP 3 C00028 BC00028  +REFP EC00028
CALL JOB:SEARCH-R1-S13D
SET P031 P006
SFTON3D P031
SMOVL C00029 BC00029 V=166.7  +MOVJ EC00029
SREFP 3 C00030 BC00030  +REFP EC00030
CALL JOB:SEARCH-R1-S13D
SET P031 P006
SFTON3D P031
SMOVL C00031 BC00031 V=166.7  +MOVJ EC00031
MOVL C00032 BC00032 V=1000.0  +MOVJ EC00032 VJ=100.00
'EndPath S3759
'Path S3760
SFTOF3D
MOVJ C00033 BC00033 VJ=100.00  +MOVJ EC00033 VJ=100.00
MOVL C00034 BC00034 V=800.0  +MOVJ EC00034 VJ=100.00
SMOVL C00035 BC00035 V=166.7  +MOVJ EC00035
SREFP 3 C00036 BC00036  +REFP EC00036
CALL JOB:SEARCH-R1-S13D
SET P032 P006
SFTON3D P032
SMOVL C00037 BC00037 V=166.7  +MOVJ EC00037
SREFP 3 C00038 BC00038  +REFP EC00038
CALL JOB:SEARCH-R1-S13D
SET P032 P006
SFTON3D P032
SMOVL C00039 BC00039 V=166.7  +MOVJ EC00039
MOVL C00040 BC00040 V=1000.0  +MOVJ EC00040 VJ=100.00
'EndPath S3760
MOVJ C00041 BC00041 VJ=100.00  +MOVJ EC00041 VJ=100.00
'
'Path S3761
SFTOF3D
MOVJ C00042 BC00042 VJ=100.00  +MOVJ EC00042 VJ=100.00
MOVL C00043 BC00043 V=800.0  +MOVJ EC00043 VJ=100.00
SMOVL C00044 BC00044 V=166.7  +MOVJ EC00044
SREFP 3 C00045 BC00045  +REFP EC00045
CALL JOB:SEARCH-R1-S13D
SET P041 P006
SFTON3D P041
SMOVL C00046 BC00046 V=166.7  +MOVJ EC00046
SREFP 3 C00047 BC00047  +REFP EC00047
CALL JOB:SEARCH-R1-S13D
SET P041 P006
SFTON3D P041
SMOVL C00048 BC00048 V=166.7  +MOVJ EC00048
SREFP 3 C00049 BC00049  +REFP EC00049
CALL JOB:SEARCH-R1-S13D
SET P041 P006
SFTON3D P041
SMOVL C00050 BC00050 V=166.7  +MOVJ EC00050
MOVL C00051 BC00051 V=1000.0  +MOVJ EC00051 VJ=100.00
'EndPath S3761
'Path S3762
SFTOF3D
MOVJ C00052 BC00052 VJ=100.00  +MOVJ EC00052 VJ=100.00
MOVL C00053 BC00053 V=800.0  +MOVJ EC00053 VJ=100.00
SMOVL C00054 BC00054 V=166.7  +MOVJ EC00054
SREFP 3 C00055 BC00055  +REFP EC00055
CALL JOB:SEARCH-R1-S13D
SET P042 P006
SFTON3D P042
SMOVL C00056 BC00056 V=166.7  +MOVJ EC00056
SREFP 3 C00057 BC00057  +REFP EC00057
CALL JOB:SEARCH-R1-S13D
SET P042 P006
SFTON3D P042
SMOVL C00058 BC00058 V=166.7  +MOVJ EC00058
MOVL C00059 BC00059 V=1000.0  +MOVJ EC00059 VJ=100.00
'EndPath S3762
MOVJ C00060 BC00060 VJ=100.00  +MOVJ EC00060 VJ=100.00
'
'Path S3763
SFTOF3D
MOVJ C00061 BC00061 VJ=100.00  +MOVJ EC00061 VJ=100.00
MOVL C00062 BC00062 V=800.0  +MOVJ EC00062 VJ=100.00
SMOVL C00063 BC00063 V=166.7  +MOVJ EC00063
SREFP 3 C00064 BC00064  +REFP EC00064
CALL JOB:SEARCH-R1-S13D
SET P051 P006
SFTON3D P051
SMOVL C00065 BC00065 V=166.7  +MOVJ EC00065
SREFP 3 C00066 BC00066  +REFP EC00066
CALL JOB:SEARCH-R1-S13D
SET P051 P006
SFTON3D P051
SMOVL C00067 BC00067 V=166.7  +MOVJ EC00067
SREFP 3 C00068 BC00068  +REFP EC00068
CALL JOB:SEARCH-R1-S13D
SET P051 P006
SFTON3D P051
SMOVL C00069 BC00069 V=166.7  +MOVJ EC00069
MOVL C00070 BC00070 V=1000.0  +MOVJ EC00070 VJ=100.00
'EndPath S3763
'Path S3764
SFTOF3D
MOVJ C00071 BC00071 VJ=100.00  +MOVJ EC00071 VJ=100.00
MOVL C00072 BC00072 V=800.0  +MOVJ EC00072 VJ=100.00
SMOVL C00073 BC00073 V=166.7  +MOVJ EC00073
SREFP 3 C00074 BC00074  +REFP EC00074
CALL JOB:SEARCH-R1-S13D
SET P052 P006
SFTON3D P052
SMOVL C00075 BC00075 V=166.7  +MOVJ EC00075
SREFP 3 C00076 BC00076  +REFP EC00076
CALL JOB:SEARCH-R1-S13D
SET P052 P006
SFTON3D P052
SMOVL C00077 BC00077 V=166.7  +MOVJ EC00077
MOVL C00078 BC00078 V=1000.0  +MOVJ EC00078 VJ=100.00
'EndPath S3764
MOVJ C00079 BC00079 VJ=100.00  +MOVJ EC00079 VJ=100.00
'
'Path S3765
SFTOF3D
MOVJ C00080 BC00080 VJ=100.00  +MOVJ EC00080 VJ=100.00
MOVL C00081 BC00081 V=800.0  +MOVJ EC00081 VJ=100.00
SMOVL C00082 BC00082 V=166.7  +MOVJ EC00082
SREFP 3 C00083 BC00083  +REFP EC00083
CALL JOB:SEARCH-R1-S13D
SET P061 P006
SFTON3D P061
SMOVL C00084 BC00084 V=166.7  +MOVJ EC00084
SREFP 3 C00085 BC00085  +REFP EC00085
CALL JOB:SEARCH-R1-S13D
SET P061 P006
SFTON3D P061
SMOVL C00086 BC00086 V=166.7  +MOVJ EC00086
SMOVL C00087 BC00087 V=166.7  +MOVJ EC00087
SREFP 3 C00088 BC00088  +REFP EC00088
CALL JOB:SEARCH-R1-S13D
SET P061 P006
SFTON3D P061
SMOVL C00089 BC00089 V=166.7  +MOVJ EC00089
MOVL C00090 BC00090 V=1000.0  +MOVJ EC00090 VJ=100.00
'EndPath S3765
'Path S3766
SFTOF3D
MOVJ C00091 BC00091 VJ=100.00  +MOVJ EC00091 VJ=100.00
MOVL C00092 BC00092 V=800.0  +MOVJ EC00092 VJ=100.00
SMOVL C00093 BC00093 V=166.7  +MOVJ EC00093
SREFP 3 C00094 BC00094  +REFP EC00094
CALL JOB:SEARCH-R1-S13D
SET P062 P006
SFTON3D P062
SMOVL C00095 BC00095 V=166.7  +MOVJ EC00095
SREFP 3 C00096 BC00096  +REFP EC00096
CALL JOB:SEARCH-R1-S13D
SET P062 P006
SFTON3D P062
SMOVL C00097 BC00097 V=166.7  +MOVJ EC00097
MOVL C00098 BC00098 V=1000.0  +MOVJ EC00098 VJ=100.00
'EndPath S3766
MOVJ C00099 BC00099 VJ=100.00  +MOVJ EC00099 VJ=100.00
'
MOVJ C00100 BC00100 VJ=100.00  +MOVJ EC00100 VJ=100.00
MOVJ C00101 BC00101 VJ=100.00  +MOVJ EC00101 VJ=100.00
'Path S3767
SFTOF3D
MOVJ C00102 BC00102 VJ=100.00  +MOVJ EC00102 VJ=100.00
MOVL C00103 BC00103 V=800.0  +MOVJ EC00103 VJ=100.00
SMOVL C00104 BC00104 V=166.7  +MOVJ EC00104
SREFP 3 C00105 BC00105  +REFP EC00105
CALL JOB:SEARCH-R1-S13D
SET P063 P006
SFTON3D P063
SMOVL C00106 BC00106 V=166.7  +MOVJ EC00106
SREFP 3 C00107 BC00107  +REFP EC00107
CALL JOB:SEARCH-R1-S13D
SET P063 P006
SFTON3D P063
SMOVL C00108 BC00108 V=166.7  +MOVJ EC00108
MOVL C00109 BC00109 V=1000.0  +MOVJ EC00109 VJ=100.00
'EndPath S3767
MOVJ C00110 BC00110 VJ=100.00  +MOVJ EC00110 VJ=100.00
MOVJ C00111 BC00111 VJ=100.00  +MOVJ EC00111 VJ=100.00
'Path S3768
SFTOF3D
MOVJ C00112 BC00112 VJ=100.00  +MOVJ EC00112 VJ=100.00
MOVL C00113 BC00113 V=800.0  +MOVJ EC00113 VJ=100.00
SMOVL C00114 BC00114 V=166.7  +MOVJ EC00114
SREFP 3 C00115 BC00115  +REFP EC00115
CALL JOB:SEARCH-R1-S13D
SET P053 P006
SFTON3D P053
SMOVL C00116 BC00116 V=166.7  +MOVJ EC00116
SREFP 3 C00117 BC00117  +REFP EC00117
CALL JOB:SEARCH-R1-S13D
SET P053 P006
SFTON3D P053
SMOVL C00118 BC00118 V=166.7  +MOVJ EC00118
MOVL C00119 BC00119 V=1000.0  +MOVJ EC00119 VJ=100.00
'EndPath S3768
MOVJ C00120 BC00120 VJ=100.00  +MOVJ EC00120 VJ=100.00
MOVJ C00121 BC00121 VJ=100.00  +MOVJ EC00121 VJ=100.00
'Path S3769
SFTOF3D
MOVJ C00122 BC00122 VJ=100.00  +MOVJ EC00122 VJ=100.00
MOVL C00123 BC00123 V=800.0  +MOVJ EC00123 VJ=100.00
SMOVL C00124 BC00124 V=166.7  +MOVJ EC00124
SREFP 3 C00125 BC00125  +REFP EC00125
CALL JOB:SEARCH-R1-S13D
SET P043 P006
SFTON3D P043
SMOVL C00126 BC00126 V=166.7  +MOVJ EC00126
SREFP 3 C00127 BC00127  +REFP EC00127
CALL JOB:SEARCH-R1-S13D
SET P043 P006
SFTON3D P043
SMOVL C00128 BC00128 V=166.7  +MOVJ EC00128
MOVL C00129 BC00129 V=1000.0  +MOVJ EC00129 VJ=100.00
'EndPath S3769
MOVJ C00130 BC00130 VJ=100.00  +MOVJ EC00130 VJ=100.00
MOVJ C00131 BC00131 VJ=100.00  +MOVJ EC00131 VJ=100.00
'Path S3770
SFTOF3D
MOVJ C00132 BC00132 VJ=100.00  +MOVJ EC00132 VJ=100.00
MOVL C00133 BC00133 V=800.0  +MOVJ EC00133 VJ=100.00
SMOVL C00134 BC00134 V=166.7  +MOVJ EC00134
SREFP 3 C00135 BC00135  +REFP EC00135
CALL JOB:SEARCH-R1-S13D
SET P033 P006
SFTON3D P033
SMOVL C00136 BC00136 V=166.7  +MOVJ EC00136
SREFP 3 C00137 BC00137  +REFP EC00137
CALL JOB:SEARCH-R1-S13D
SET P033 P006
SFTON3D P033
SMOVL C00138 BC00138 V=166.7  +MOVJ EC00138
MOVL C00139 BC00139 V=1000.0  +MOVJ EC00139 VJ=100.00
'EndPath S3770
MOVJ C00140 BC00140 VJ=100.00  +MOVJ EC00140 VJ=100.00
MOVJ C00141 BC00141 VJ=100.00  +MOVJ EC00141 VJ=100.00
'Path S3771
SFTOF3D
MOVJ C00142 BC00142 VJ=100.00  +MOVJ EC00142 VJ=100.00
MOVL C00143 BC00143 V=800.0  +MOVJ EC00143 VJ=100.00
SMOVL C00144 BC00144 V=166.7  +MOVJ EC00144
SREFP 3 C00145 BC00145  +REFP EC00145
CALL JOB:SEARCH-R1-S13D
SET P023 P006
SFTON3D P023
SMOVL C00146 BC00146 V=166.7  +MOVJ EC00146
SREFP 3 C00147 BC00147  +REFP EC00147
CALL JOB:SEARCH-R1-S13D
SET P023 P006
SFTON3D P023
SMOVL C00148 BC00148 V=166.7  +MOVJ EC00148
MOVL C00149 BC00149 V=1000.0  +MOVJ EC00149 VJ=100.00
'EndPath S3771
MOVJ C00150 BC00150 VJ=100.00  +MOVJ EC00150 VJ=100.00
'
'
'
'Path W3772
SFTOF3D
SFTON3D P043
MOVJ C00151 BC00151 VJ=100.00  +MOVJ EC00151 VJ=100.00
SMOVL C00152 BC00152 V=800.0  +MOVJ EC00152
SMOVL C00153 BC00153 V=166.7 PL=0  +MOVJ EC00153
MACRO1 MJ#(0) ARGF9
ARCON
SMOVL C00154 BC00154 V=10.0  +MOVJ EC00154
SMOVL C00155 BC00155 V=10.0  +MOVJ EC00155
SMOVL C00156 BC00156 V=10.0  +MOVJ EC00156
SMOVL C00157 BC00157 V=10.0  +MOVJ EC00157
SMOVL C00158 BC00158 V=10.0  +MOVJ EC00158
SMOVL C00159 BC00159 V=10.0  +MOVJ EC00159
ARCOF
SMOVL C00160 BC00160 V=800.0  +MOVJ EC00160
SMOVL C00161 BC00161 V=1000.0  +MOVJ EC00161
SFTOF3D
'EndPath W3772
MOVJ C00162 BC00162 VJ=100.00  +MOVJ EC00162 VJ=100.00
MOVJ C00163 BC00163 VJ=100.00  +MOVJ EC00163 VJ=100.00
'Path W3773
SFTOF3D
SFTON3D P023
MOVJ C00164 BC00164 VJ=100.00  +MOVJ EC00164 VJ=100.00
SMOVL C00165 BC00165 V=800.0  +MOVJ EC00165
SMOVL C00166 BC00166 V=166.7 PL=0  +MOVJ EC00166
ARCON
SMOVL C00167 BC00167 V=10.0  +MOVJ EC00167
SMOVL C00168 BC00168 V=10.0  +MOVJ EC00168
SMOVL C00169 BC00169 V=10.0  +MOVJ EC00169
SMOVL C00170 BC00170 V=10.0  +MOVJ EC00170
SMOVL C00171 BC00171 V=10.0  +MOVJ EC00171
ARCOF
SMOVL C00172 BC00172 V=800.0  +MOVJ EC00172
SMOVL C00173 BC00173 V=1000.0  +MOVJ EC00173
SFTOF3D
'EndPath W3773
MOVJ C00174 BC00174 VJ=100.00  +MOVJ EC00174 VJ=100.00
MOVJ C00175 BC00175 VJ=100.00  +MOVJ EC00175 VJ=100.00
'Path W3774
SFTOF3D
SFTON3D P063
MOVJ C00176 BC00176 VJ=100.00  +MOVJ EC00176 VJ=100.00
SMOVL C00177 BC00177 V=800.0  +MOVJ EC00177
SMOVL C00178 BC00178 V=166.7 PL=0  +MOVJ EC00178
ARCON
SMOVL C00179 BC00179 V=10.0  +MOVJ EC00179
SMOVL C00180 BC00180 V=10.0  +MOVJ EC00180
SMOVL C00181 BC00181 V=10.0  +MOVJ EC00181
SMOVL C00182 BC00182 V=10.0  +MOVJ EC00182
SMOVL C00183 BC00183 V=10.0  +MOVJ EC00183
SMOVL C00184 BC00184 V=10.0  +MOVJ EC00184
ARCOF
SMOVL C00185 BC00185 V=800.0  +MOVJ EC00185
SMOVL C00186 BC00186 V=1000.0  +MOVJ EC00186
SFTOF3D
'EndPath W3774
MOVJ C00187 BC00187 VJ=100.00  +MOVJ EC00187 VJ=100.00
MOVJ C00188 BC00188 VJ=100.00  +MOVJ EC00188 VJ=100.00
'Path W3775
SFTOF3D
SFTON3D P033
MOVJ C00189 BC00189 VJ=100.00  +MOVJ EC00189 VJ=100.00
SMOVL C00190 BC00190 V=800.0  +MOVJ EC00190
SMOVL C00191 BC00191 V=166.7 PL=0  +MOVJ EC00191
ARCON
SMOVL C00192 BC00192 V=10.0  +MOVJ EC00192
SMOVL C00193 BC00193 V=10.0  +MOVJ EC00193
SMOVL C00194 BC00194 V=10.0  +MOVJ EC00194
SMOVL C00195 BC00195 V=10.0  +MOVJ EC00195
SMOVL C00196 BC00196 V=10.0  +MOVJ EC00196
ARCOF
SMOVL C00197 BC00197 V=800.0  +MOVJ EC00197
SMOVL C00198 BC00198 V=1000.0  +MOVJ EC00198
SFTOF3D
'EndPath W3775
MOVJ C00199 BC00199 VJ=100.00  +MOVJ EC00199 VJ=100.00
MOVJ C00200 BC00200 VJ=100.00  +MOVJ EC00200 VJ=100.00
'Path W3776
SFTOF3D
SFTON3D P053
MOVJ C00201 BC00201 VJ=100.00  +MOVJ EC00201 VJ=100.00
SMOVL C00202 BC00202 V=800.0  +MOVJ EC00202
SMOVL C00203 BC00203 V=166.7 PL=0  +MOVJ EC00203
ARCON
SMOVL C00204 BC00204 V=10.0  +MOVJ EC00204
SMOVL C00205 BC00205 V=10.0  +MOVJ EC00205
SMOVL C00206 BC00206 V=10.0  +MOVJ EC00206
SMOVL C00207 BC00207 V=10.0  +MOVJ EC00207
SMOVL C00208 BC00208 V=10.0  +MOVJ EC00208
ARCOF
SMOVL C00209 BC00209 V=800.0  +MOVJ EC00209
SMOVL C00210 BC00210 V=1000.0  +MOVJ EC00210
SFTOF3D
'EndPath W3776
MOVJ C00211 BC00211 VJ=100.00  +MOVJ EC00211 VJ=100.00
MOVJ C00212 BC00212 VJ=100.00  +MOVJ EC00212 VJ=100.00
MOVJ C00213 BC00213 VJ=100.00  +MOVJ EC00213 VJ=100.00
'
MOVJ C00214 BC00214 VJ=100.00  +MOVJ EC00214 VJ=100.00
'Path W3777
SFTOF3D
SFTON3D P042
MOVJ C00215 BC00215 VJ=100.00  +MOVJ EC00215 VJ=100.00
SMOVL C00216 BC00216 V=800.0  +MOVJ EC00216
SMOVL C00217 BC00217 V=166.7 PL=0  +MOVJ EC00217
ARCON
SMOVL C00218 BC00218 V=10.0  +MOVJ EC00218
SMOVL C00219 BC00219 V=10.0  +MOVJ EC00219
SMOVL C00220 BC00220 V=10.0  +MOVJ EC00220
SMOVL C00221 BC00221 V=10.0  +MOVJ EC00221
SMOVL C00222 BC00222 V=10.0  +MOVJ EC00222
ARCOF
SMOVL C00223 BC00223 V=800.0  +MOVJ EC00223
SMOVL C00224 BC00224 V=1000.0  +MOVJ EC00224
SFTOF3D
'EndPath W3777
'Path W3778
SFTOF3D
SFTON3D P041
MOVJ C00225 BC00225 VJ=100.00  +MOVJ EC00225 VJ=100.00
SMOVL C00226 BC00226 V=800.0  +MOVJ EC00226
SMOVL C00227 BC00227 V=166.7 PL=0  +MOVJ EC00227
ARCON
SMOVL C00228 BC00228 V=10.0  +MOVJ EC00228
SMOVL C00229 BC00229 V=10.0  +MOVJ EC00229
SMOVL C00230 BC00230 V=10.0  +MOVJ EC00230
SMOVL C00231 BC00231 V=10.0  +MOVJ EC00231
ARCOF
SMOVL C00232 BC00232 V=800.0  +MOVJ EC00232
SMOVL C00233 BC00233 V=1000.0  +MOVJ EC00233
SFTOF3D
'EndPath W3778
'Path W3779
SFTOF3D
SFTON3D P041
MOVJ C00234 BC00234 VJ=100.00  +MOVJ EC00234 VJ=100.00
SMOVL C00235 BC00235 V=800.0  +MOVJ EC00235
SMOVL C00236 BC00236 V=166.7 PL=0  +MOVJ EC00236
ARCON
SMOVL C00237 BC00237 V=10.0  +MOVJ EC00237
SMOVL C00238 BC00238 V=10.0  +MOVJ EC00238
SMOVL C00239 BC00239 V=10.0  +MOVJ EC00239
ARCOF
SMOVL C00240 BC00240 V=800.0  +MOVJ EC00240
SMOVL C00241 BC00241 V=1000.0  +MOVJ EC00241
SFTOF3D
'EndPath W3779
MOVJ C00242 BC00242 VJ=100.00  +MOVJ EC00242 VJ=100.00
'
'
MOVJ C00243 BC00243 VJ=100.00  +MOVJ EC00243 VJ=100.00
'Path W3780
SFTOF3D
SFTON3D P022
MOVJ C00244 BC00244 VJ=100.00  +MOVJ EC00244 VJ=100.00
SMOVL C00245 BC00245 V=800.0  +MOVJ EC00245
SMOVL C00246 BC00246 V=166.7 PL=0  +MOVJ EC00246
ARCON
SMOVL C00247 BC00247 V=10.0  +MOVJ EC00247
SMOVL C00248 BC00248 V=10.0  +MOVJ EC00248
SMOVL C00249 BC00249 V=10.0  +MOVJ EC00249
ARCOF
SMOVL C00250 BC00250 V=800.0  +MOVJ EC00250
SMOVL C00251 BC00251 V=1000.0  +MOVJ EC00251
SFTOF3D
'EndPath W3780
'Path W3781
SFTOF3D
SFTON3D P021
MOVJ C00252 BC00252 VJ=100.00  +MOVJ EC00252 VJ=100.00
SMOVL C00253 BC00253 V=800.0  +MOVJ EC00253
SMOVL C00254 BC00254 V=166.7 PL=0  +MOVJ EC00254
ARCON
SMOVL C00255 BC00255 V=10.0  +MOVJ EC00255
SMOVL C00256 BC00256 V=10.0  +MOVJ EC00256
SMOVL C00257 BC00257 V=10.0  +MOVJ EC00257
SMOVL C00258 BC00258 V=10.0  +MOVJ EC00258
ARCOF
SMOVL C00259 BC00259 V=800.0  +MOVJ EC00259
SMOVL C00260 BC00260 V=1000.0  +MOVJ EC00260
SFTOF3D
'EndPath W3781
'Path W3782
SFTOF3D
SFTON3D P021
MOVJ C00261 BC00261 VJ=100.00  +MOVJ EC00261 VJ=100.00
SMOVL C00262 BC00262 V=800.0  +MOVJ EC00262
SMOVL C00263 BC00263 V=166.7 PL=0  +MOVJ EC00263
ARCON
SMOVL C00264 BC00264 V=10.0  +MOVJ EC00264
SMOVL C00265 BC00265 V=10.0  +MOVJ EC00265
SMOVL C00266 BC00266 V=10.0  +MOVJ EC00266
ARCOF
SMOVL C00267 BC00267 V=800.0  +MOVJ EC00267
SMOVL C00268 BC00268 V=1000.0  +MOVJ EC00268
SFTOF3D
'EndPath W3782
MOVJ C00269 BC00269 VJ=100.00  +MOVJ EC00269 VJ=100.00
'
'
MOVJ C00270 BC00270 VJ=100.00  +MOVJ EC00270 VJ=100.00
'Path W3783
SFTOF3D
SFTON3D P062
MOVJ C00271 BC00271 VJ=100.00  +MOVJ EC00271 VJ=100.00
SMOVL C00272 BC00272 V=800.0  +MOVJ EC00272
SMOVL C00273 BC00273 V=166.7 PL=0  +MOVJ EC00273
ARCON
SMOVL C00274 BC00274 V=10.0  +MOVJ EC00274
SMOVL C00275 BC00275 V=10.0  +MOVJ EC00275
SMOVL C00276 BC00276 V=10.0  +MOVJ EC00276
SMOVL C00277 BC00277 V=10.0  +MOVJ EC00277
SMOVL C00278 BC00278 V=10.0  +MOVJ EC00278
ARCOF
SMOVL C00279 BC00279 V=800.0  +MOVJ EC00279
SMOVL C00280 BC00280 V=1000.0  +MOVJ EC00280
SFTOF3D
'EndPath W3783
'Path W3784
SFTOF3D
SFTON3D P061
MOVJ C00281 BC00281 VJ=100.00  +MOVJ EC00281 VJ=100.00
SMOVL C00282 BC00282 V=800.0  +MOVJ EC00282
SMOVL C00283 BC00283 V=166.7 PL=0  +MOVJ EC00283
ARCON
SMOVL C00284 BC00284 V=10.0  +MOVJ EC00284
SMOVL C00285 BC00285 V=10.0  +MOVJ EC00285
SMOVL C00286 BC00286 V=10.0  +MOVJ EC00286
SMOVL C00287 BC00287 V=10.0  +MOVJ EC00287
ARCOF
SMOVL C00288 BC00288 V=800.0  +MOVJ EC00288
SMOVL C00289 BC00289 V=1000.0  +MOVJ EC00289
SFTOF3D
'EndPath W3784
'Path W3785
SFTOF3D
SFTON3D P061
MOVJ C00290 BC00290 VJ=100.00  +MOVJ EC00290 VJ=100.00
SMOVL C00291 BC00291 V=800.0  +MOVJ EC00291
SMOVL C00292 BC00292 V=166.7 PL=0  +MOVJ EC00292
ARCON
SMOVL C00293 BC00293 V=10.0  +MOVJ EC00293
SMOVL C00294 BC00294 V=10.0  +MOVJ EC00294
SMOVL C00295 BC00295 V=10.0  +MOVJ EC00295
ARCOF
SMOVL C00296 BC00296 V=800.0  +MOVJ EC00296
SMOVL C00297 BC00297 V=1000.0  +MOVJ EC00297
SFTOF3D
'EndPath W3785
MOVJ C00298 BC00298 VJ=100.00  +MOVJ EC00298 VJ=100.00
'
'
MOVJ C00299 BC00299 VJ=100.00  +MOVJ EC00299 VJ=100.00
'Path W3786
SFTOF3D
SFTON3D P032
MOVJ C00300 BC00300 VJ=100.00  +MOVJ EC00300 VJ=100.00
SMOVL C00301 BC00301 V=800.0  +MOVJ EC00301
SMOVL C00302 BC00302 V=166.7 PL=0  +MOVJ EC00302
ARCON
SMOVL C00303 BC00303 V=10.0  +MOVJ EC00303
SMOVL C00304 BC00304 V=10.0  +MOVJ EC00304
SMOVL C00305 BC00305 V=10.0  +MOVJ EC00305
SMOVL C00306 BC00306 V=10.0  +MOVJ EC00306
SMOVL C00307 BC00307 V=10.0  +MOVJ EC00307
ARCOF
SMOVL C00308 BC00308 V=800.0  +MOVJ EC00308
SMOVL C00309 BC00309 V=1000.0  +MOVJ EC00309
SFTOF3D
'EndPath W3786
'Path W3787
SFTOF3D
SFTON3D P031
MOVJ C00310 BC00310 VJ=100.00  +MOVJ EC00310 VJ=100.00
SMOVL C00311 BC00311 V=800.0  +MOVJ EC00311
SMOVL C00312 BC00312 V=166.7 PL=0  +MOVJ EC00312
ARCON
SMOVL C00313 BC00313 V=10.0  +MOVJ EC00313
SMOVL C00314 BC00314 V=10.0  +MOVJ EC00314
SMOVL C00315 BC00315 V=10.0  +MOVJ EC00315
SMOVL C00316 BC00316 V=10.0  +MOVJ EC00316
ARCOF
SMOVL C00317 BC00317 V=800.0  +MOVJ EC00317
SMOVL C00318 BC00318 V=1000.0  +MOVJ EC00318
SFTOF3D
'EndPath W3787
'Path W3788
SFTOF3D
SFTON3D P031
MOVJ C00319 BC00319 VJ=100.00  +MOVJ EC00319 VJ=100.00
SMOVL C00320 BC00320 V=800.0  +MOVJ EC00320
SMOVL C00321 BC00321 V=166.7 PL=0  +MOVJ EC00321
ARCON
SMOVL C00322 BC00322 V=10.0  +MOVJ EC00322
SMOVL C00323 BC00323 V=10.0  +MOVJ EC00323
SMOVL C00324 BC00324 V=10.0  +MOVJ EC00324
ARCOF
SMOVL C00325 BC00325 V=800.0  +MOVJ EC00325
SMOVL C00326 BC00326 V=1000.0  +MOVJ EC00326
SFTOF3D
'EndPath W3788
MOVJ C00327 BC00327 VJ=100.00  +MOVJ EC00327 VJ=100.00
'
'
MOVJ C00328 BC00328 VJ=100.00  +MOVJ EC00328 VJ=100.00
'Path W3789
SFTOF3D
SFTON3D P052
MOVJ C00329 BC00329 VJ=100.00  +MOVJ EC00329 VJ=100.00
SMOVL C00330 BC00330 V=800.0  +MOVJ EC00330
SMOVL C00331 BC00331 V=166.7 PL=0  +MOVJ EC00331
ARCON
SMOVL C00332 BC00332 V=10.0  +MOVJ EC00332
SMOVL C00333 BC00333 V=10.0  +MOVJ EC00333
SMOVL C00334 BC00334 V=10.0  +MOVJ EC00334
ARCOF
SMOVL C00335 BC00335 V=800.0  +MOVJ EC00335
SMOVL C00336 BC00336 V=1000.0  +MOVJ EC00336
SFTOF3D
'EndPath W3789
'Path W3790
SFTOF3D
SFTON3D P051
MOVJ C00337 BC00337 VJ=100.00  +MOVJ EC00337 VJ=100.00
SMOVL C00338 BC00338 V=800.0  +MOVJ EC00338
SMOVL C00339 BC00339 V=166.7 PL=0  +MOVJ EC00339
ARCON
SMOVL C00340 BC00340 V=10.0  +MOVJ EC00340
SMOVL C00341 BC00341 V=10.0  +MOVJ EC00341
SMOVL C00342 BC00342 V=10.0  +MOVJ EC00342
SMOVL C00343 BC00343 V=10.0  +MOVJ EC00343
ARCOF
SMOVL C00344 BC00344 V=800.0  +MOVJ EC00344
SMOVL C00345 BC00345 V=1000.0  +MOVJ EC00345
SFTOF3D
'EndPath W3790
'Path W3791
SFTOF3D
SFTON3D P051
MOVJ C00346 BC00346 VJ=100.00  +MOVJ EC00346 VJ=100.00
SMOVL C00347 BC00347 V=800.0  +MOVJ EC00347
SMOVL C00348 BC00348 V=166.7 PL=0  +MOVJ EC00348
ARCON
SMOVL C00349 BC00349 V=10.0  +MOVJ EC00349
SMOVL C00350 BC00350 V=10.0  +MOVJ EC00350
SMOVL C00351 BC00351 V=10.0  +MOVJ EC00351
ARCOF
SMOVL C00352 BC00352 V=800.0  +MOVJ EC00352
SMOVL C00353 BC00353 V=1000.0  +MOVJ EC00353
SFTOF3D
'EndPath W3791
MOVJ C00354 BC00354 VJ=100.00  +MOVJ EC00354 VJ=100.00
'
MOVJ C00355 BC00355 VJ=100.00  +MOVJ EC00355 VJ=100.00
END
